FUNCTION_BLOCK FB_Modulo
VAR_INPUT
	fModIn1:		INT;
	fModIn2:		INT;
END_VAR
VAR_OUTPUT
	fModOut:	INT;
END_VAR
VAR
END_VAR

fModOut:= fModIn1 MOD fModIn2;

END_FUNCTION_BLOCK

(* stored: Version 1.1.0.1, ProductVersion 3.1.4024.3
   POU FB_Modulo: Id {5154f507-5910-41fc-ab44-378a007bd29c}, SpecialFunc None *)
